FUNCTION_BLOCK FB_Separator
VAR_INPUT
	bEnable : BOOL; 	// start/stops the functionblock
	bExecute: BOOL; 	// Ejects 1 flask if true
	bErrorReset: BOOL;	//Reset Error 
	
	bSensor1 : BOOL; //Hardware Sensor 1
	bSensor2 : BOOL; //Hardware Sensor 2
	bSensor3 : BOOL; //Hardware Sensor 3
END_VAR
VAR_OUTPUT
	bR1AKT1 : BOOL; //Relais 1 Aktor 1 (Schieber oben)
	bR2AKT1 : BOOL; //Relais 2 Aktor 1
	bR1AKT2 : BOOL; //Relais 1 Aktor 2 (Schieber unten)
	bR2AKT2 : BOOL; //Relais 2 Aktor 2
	
	bNoBottle		: BOOL;		//Keine Flasche vorhanden
	bWrongBottle	: BOOL; //Falsche oder gedrehte Flasche vorhanden
	
	eStatus : State := State.Off;
END_VAR
VAR
	timer : TON; //Timer to make sure, that the flask has cleared the slope
	eState : StateSeparator := StateSeparator.Off;
END_VAR

CASE eState OF
StateSeparator.Off:
	eStatus := State.Off;
	bR1AKT1 := TRUE;	//Eingefahren oben
	bR2AKT1 := FALSE;	//Eingefahren oben
	
	bR1AKT2 := FALSE;	//Eingefahren unten
	bR2AKT2 := TRUE;	//Eingefahren unten

	IF bEnable	THEN
		eState := StateSeparator.Init;
	END_IF
	
StateSeparator.Init:
	
	eStatus := State.Busy; //Beschaeftigt Signallampe

	bR1AKT1 := FALSE; //Ausgefahren oben
	bR2AKT1 := TRUE;
	
	bR1AKT2 := FALSE; //Eingefahren unten
	bR2AKT2 := TRUE;

	
	IF bSensor1 THEN
		eState := StateSeparator.Init_Wait;	//Zustandswechsel sobald Sensor Flasche zwischen Schiebern sieht
	END_IF	
	
StateSeparator.Init_Wait:
	timer(IN := TRUE, PT := T#1000MS); //Timer wartet bis Flasche sicher zum Stehen kommt
	
	IF timer.Q THEN
		timer(IN := FALSE);
		eState := StateSeparator.Ready; //Zustand Ready nach Timer
	END_IF
	
StateSeparator.Ready:
	eStatus := State.Ready; //Zustand Ready Signallampe

	bR1AKT1 := TRUE;	//Eingefahren oben
	bR2AKT1 := FALSE;	//Eingefahren oben
	
	bR1AKT2 := FALSE;	//Eingefahren unten
	bR2AKT2 := TRUE;	//Eingefahren unten
	
	IF bExecute THEN
		eState := StateSeparator.Eject_Wait_1; //Auswerfen sobald Exceute TRUE
	END_IF

StateSeparator.Eject_Wait_1:	// Warten bis Schieber oben ganz geschlossen ist
		eStatus := State.Busy; //Zustand Busy Signallampe
	
		timer(IN := TRUE, PT := T#2500MS); //Timer auf 2,5 S eingestellt
	
	IF timer.Q THEN
		timer(IN := FALSE);
		eState := StateSeparator.Eject; //Zustand bereit nach Timer
	END_IF
	
StateSeparator.Eject:	//Auswerfen der unteren Flasche
	bR1AKT2 := TRUE;	//Lässt Flaschen auf Band ab durch Öffnen des unteren Schiebers
	bR2AKT2 := FALSE;
	
	IF NOT bSensor1 THEN
		eState := StateSeparator.Eject_Wait_2; 
	END_IF
	
StateSeparator.Eject_Wait_2:	// Warten bis Flasche durch Förderband weit genug von Schieber wegtransportiert
	eStatus := State.Done;
	timer(IN := TRUE, PT := T#4000MS); //Timer auf 4 S eingestellt
	
	IF timer.Q THEN
		timer(IN := FALSE);
		eState := StateSeparator.Done_Wait; 
	END_IF 
	
StateSeparator.Done_Wait: // Schließen des unteren Schiebers und Warten bis komplettt geschlossen
	bR1AKT2 := FALSE;	//Eingefahren unten
	bR2AKT2 := TRUE;	//Eingefahren unten
	
	timer(IN := TRUE, PT := T#3000MS); //Timer wartet bis Schieber geschlossen ist
	
	IF timer.Q THEN
		timer(IN := FALSE);
		eState := StateSeparator.Done; 
	END_IF	
	
StateSeparator.Done:	//Vereinzelungsvorgang abgeschlossen
	
	IF NOT bExecute THEN
		eState := StateSeparator.Init;
	END_IF

END_CASE

END_FUNCTION_BLOCK

(* stored: Version 1.1.0.1, ProductVersion 3.1.4024.10
   POU FB_Separator: Id {91946f14-5ef9-4883-993a-962cda20c177}, SpecialFunc None *)
